// TIA Portal V17 export
// export: Created 2025-03-05T08:01:44.1026201Z, ExportSetting WithDefaults, DisplayName Totally Integrated Automation Portal, DisplayVersion V17 Update 8, DisplayName TIA Portal Openness, DisplayVersion V17 Update 8, DisplayName TIA Portal Version Control Interface, DisplayVersion V17, DisplayName SINAMICS Startdrive Advanced, DisplayVersion V17 SP2, DisplayName SINAMICS Startdrive G110M, G120, G120C, G120D, G120P, G115D, DisplayVersion V17 SP2, DisplayName SINAMICS Startdrive G130, G150, S120, S150, SINAMICS MV, S210, DisplayVersion V17 SP2, DisplayName STEP 7 Professional, DisplayVersion V17 Update 8, DisplayName SINUMERIK ONE STEP 7 Toolbox, DisplayVersion V17 Update 12, DisplayName SINUMERIK 840D sl STEP 7 Toolbox, DisplayVersion V17 Update 12, DisplayName STEP 7 Safety, DisplayVersion V17 Update 6, DisplayName WinCC Advanced, DisplayVersion V17 Update 8
DATA_BLOCK "DB7210_WORKPIECE_F1_COUNT"   // DB7210
{ DB_Accessible_From_OPC_UA := 'FALSE' }
// stored: AutoNumber false, DBAccessibleFromOPCUA false, DBAccessibleFromWebserver true, InstanceOfName LTLP_WorkpieceCount, InstanceOfType FB
"LTLP_WorkpieceCount"
   // VAR_INPUT
   //    MACHINING_UNIT : Int;
   //    COUNT_START : Bool;
   //    RESET_WORKPIECETYPE : Word;
   // END_VAR
   // VAR_OUTPUT
   //    ERROR : Word;
   // END_VAR
   // VAR_IN_OUT
   //    RESET_WHOLE : Bool;
   //    RESET_DAY : Bool;
   //    RESET_SHIFT : Bool;
   //    HMI_DB : "LTLP_typeHmiProInterface";
   //    EXTERNAL_COUNTER_DB : Variant;
   // END_VAR
   // VAR
   //    typeCount : Int;
   //    loopTypeWorked : Int;
   //    lowerBoundExternal : Int;
   //    upperBoundExternal : Int;
   //    countOfElemExternal : Int;
   //    wholeCount : DWord;
   //    wholeCountNIO : Word;
   //    dayCount : Word;
   //    dayCountNIO : Word;
   //    shiftCount : Word;
   //    shiftCountNIO : Word;
   //    fpCount : Bool;
   //    fpResetWhole : Bool;
   //    fpResetDay : Bool;
   //    fpResetShift : Bool;
   //    fpResetCounters : Bool;
   //    fpBuildSummaryCounter : Bool;
   //    buildSummaryRun : Bool;
   //    externalCounter { S7_SetPoint := 'True'} : "LTLP_typeWorkpieceCount";
   // END_VAR
BEGIN
END_DATA_BLOCK
